(* IEC 61131-3 sources: repolevel_ST_code_completion/dataset/project_code/VisuElements/FUN, 3 files *)

(* ---- RotationCalculation.st ---- *)
FUNCTION RotationCalculation : BOOL
VAR_INPUT
    rCenterX : REAL;    (* X coordinate of rotation center *)
    rCenterY : REAL;    (* Y coordinate of rotation center *)
    rAngle : REAL;      (* Rotation angle in degrees *)
    rPointX : REAL;     (* X coordinate of point to rotate *)
    rPointY : REAL;     (* Y coordinate of point to rotate *)
END_VAR

VAR_OUTPUT
    rRotatedX : REAL;   (* X coordinate after rotation *)
    rRotatedY : REAL;   (* Y coordinate after rotation *)
END_VAR

VAR
    rRadians : REAL;
    rCos : REAL;
    rSin : REAL;
    rTranslatedX : REAL;
    rTranslatedY : REAL;
END_VAR

(* Convert angle from degrees to radians *)
rRadians := rAngle * 3.14159 / 180.0;

(* Calculate sine and cosine *)
rCos := COS(rRadians);
rSin := SIN(rRadians);

(* Translate point to origin (relative to center) *)
rTranslatedX := rPointX - rCenterX;
rTranslatedY := rPointY - rCenterY;

(* Apply rotation matrix *)
rRotatedX := rTranslatedX * rCos - rTranslatedY * rSin;
rRotatedY := rTranslatedX * rSin + rTranslatedY * rCos;

(* Translate back to original position *)
rRotatedX := rRotatedX + rCenterX;
rRotatedY := rRotatedY + rCenterY;

RotationCalculation := TRUE;  (* Return success *)

(* ---- MouseEventHandler.st ---- *)
FUNCTION_BLOCK MouseEventHandler
VAR_INPUT
    xLeftClick : BOOL;      (* Left mouse button click *)
    xRightClick : BOOL;     (* Right mouse button click *)
    xMiddleClick : BOOL;    (* Middle mouse button click *)
    xMouseMove : BOOL;      (* Mouse movement detected *)
    rMouseX : REAL;         (* Current mouse X position *)
    rMouseY : REAL;         (* Current mouse Y position *)
    tDblClickTime : TIME := T#300MS;  (* Double click timeout *)
END_VAR

VAR_OUTPUT
    eMouseEvent : INT;      (* Event type: 0=None, 1=SingleClick, 2=DoubleClick, 3=RightClick, 4=MiddleClick *)
    rEventX : REAL;         (* X position where event occurred *)
    rEventY : REAL;         (* Y position where event occurred *)
    xEventActive : BOOL;    (* TRUE when an event is active *)
END_VAR

VAR
    LeftClickTimer : TON;
    xLeftClickOld : BOOL;
    iClickCount : INT := 0;
    xEventProcessed : BOOL := FALSE;
END_VAR

(* Reset event state *)
eMouseEvent := 0;
xEventActive := FALSE;

(* Handle left click events (single/double click) *)
IF xLeftClick AND NOT xLeftClickOld THEN
    (* First click detected *)
    IF iClickCount = 0 THEN
        LeftClickTimer(IN:=TRUE, PT:=tDblClickTime);
        iClickCount := 1;
    ELSE
        (* Second click within time window *)
        LeftClickTimer(IN:=FALSE);
        eMouseEvent := 2; (* Double click *)
        rEventX := rMouseX;
        rEventY := rMouseY;
        xEventActive := TRUE;
        iClickCount := 0;
        xEventProcessed := TRUE;
    END_IF
ELSIF NOT xLeftClick AND xLeftClickOld THEN
    (* Left button released *)
    IF iClickCount = 1 AND NOT xEventProcessed THEN
        LeftClickTimer();
        IF NOT LeftClickTimer.Q THEN
            (* Still waiting for potential double click *)
            (* Will be handled by timer logic below *)
        END_IF
    END_IF
END_IF

(* Check for double click timeout *)
IF LeftClickTimer.Q AND iClickCount = 1 AND NOT xEventProcessed THEN
    (* Timeout - single click confirmed *)
    LeftClickTimer(IN:=FALSE);
    eMouseEvent := 1; (* Single click *)
    rEventX := rMouseX;
    rEventY := rMouseY;
    xEventActive := TRUE;
    iClickCount := 0;
END_IF

(* Handle right click *)
IF xRightClick AND NOT xEventProcessed THEN
    eMouseEvent := 3; (* Right click *)
    rEventX := rMouseX;
    rEventY := rMouseY;
    xEventActive := TRUE;
    xEventProcessed := TRUE;
END_IF

(* Handle middle click *)
IF xMiddleClick AND NOT xEventProcessed THEN
    eMouseEvent := 4; (* Middle click *)
    rEventX := rMouseX;
    rEventY := rMouseY;
    xEventActive := TRUE;
    xEventProcessed := TRUE;
END_IF

(* Update old states *)
xLeftClickOld := xLeftClick;

(* Reset processed flag for next cycle *)
xEventProcessed := FALSE;

(* ---- NodeExpandCollapse.st ---- *)
FUNCTION_BLOCK NodeExpandCollapse
VAR_INPUT
    xNodeClick : BOOL;  (* Input signal for node click *)
    tDblClickTime : TIME := T#500MS;  (* Time to wait for double click *)
END_VAR

VAR_OUTPUT
    xNodeExpand : BOOL;  (* Output: TRUE when node is expanded *)
    xNodeSelected : BOOL; (* Output: TRUE when node is selected *)
END_VAR

VAR
    NodeDblClick : TON;
    xNodeClickOld : BOOL;
    iNodeState : INT := 1;
END_VAR

(* This function block handles double-click expansion/collapse of a node *)

CASE iNodeState OF

    1: (* Wait for first click *)
        IF xNodeClick AND NOT xNodeClickOld THEN
            NodeDblClick(IN:=TRUE, PT:=tDblClickTime);
            iNodeState := 2;
            xNodeSelected := TRUE;
        END_IF

    2: (* Wait for second click or timeout *)
        NodeDblClick();
        IF NodeDblClick.Q THEN
            (* Timeout - single click, reset *)
            NodeDblClick(IN:=FALSE);
            xNodeClickOld := FALSE;
            iNodeState := 1;
            xNodeSelected := FALSE;
        ELSIF NOT xNodeClick AND xNodeClickOld THEN
            (* Second click detected - toggle expansion *)
            NodeDblClick(IN:=FALSE);
            xNodeExpand := NOT xNodeExpand;
            iNodeState := 1;
            xNodeSelected := FALSE;
        END_IF
END_CASE

xNodeClickOld := xNodeClick;
